// TIA Portal V19 export
TYPE "dtStepSP"
   STRUCT
      "type" { S7_SetPoint := 'True'} : Int;   // Type of step ending condition (0=time scanning, 1=condition scanning, 2=both)
      next { S7_SetPoint := 'True'} : Int;   // Next step number (when required to end leave that 0)
      timeStep { S7_SetPoint := 'True'} : "dtTimerArguments";   // Step timer arguments
      timeOut { S7_SetPoint := 'True'} : "dtTimerArguments";   // Timeout scanner arguments
   END_STRUCT;
END_TYPE
